TYPE ST_PRINTER_IN :
STRUCT

	bSystemReset			: BOOL;			(* set TRUE to send SystemReset command to printer *)
	bSendCommand		: BOOL;			(* set TRUE to send command to printer *)
	sCommand				: T_LongSTRING;	(* command to be sent to the printer *)

END_STRUCT
END_TYPE

(* stored: Version 1.1.0.1, ProductVersion 3.1.4024.15
   DUT ST_PRINTER_IN: Id {e425f444-ded7-445a-9143-db6d98072374} *)
